// TwinCAT 3 PLC project Simulation_PLC
// ProgramVersion: 3.1.4026.18
// libraries:
//   Tc2_Standard, * (Beckhoff Automation GmbH)
//   Tc2_System, * (Beckhoff Automation GmbH)
//   Tc2_TcpIp, * (Beckhoff Automation GmbH)
//   Tc3_Module, * (Beckhoff Automation GmbH)
// project tree:
//   DUTs/ADS2ROS2/ ST_Pose.TcDUT
//   DUTs/Control/ E_RemoteMode.TcDUT, ST_Control.TcDUT, ST_ControlComau.TcDUT, ST_ControlStewart.TcDUT, ST_ControlWinch.TcDUT
//   DUTs/Feedback/ ST_Feedback.TcDUT, ST_FeedbackComau.TcDUT, ST_FeedbackLeica.TcDUT, ST_FeedbackMru.TcDUT, ST_FeedbackQualisys.TcDUT, ST_FeedbackStewart.TcDUT, ST_FeedbackWinch.TcDUT
//   DUTs/QualisysRT/Components/ ST_3DMarkerPositionNoLabel.TcDUT, ST_3DMarkerPositionNoLabelComponent.TcDUT, ST_RT6D.TcDUT, ST_RT6DComponent.TcDUT, ST_TxHmiQualisys.TcDUT
//   DUTs/QualisysRT/ E_ComponentType.TcDUT, ST_RTComponentData.TcDUT, ST_RTDataQRTPacket.TcDUT
//   DUTs/ ST_RxUdpRemote.TcDUT
//   / PlcTask.TcTTO
//   POUs/ MAIN.TcPOU
//   UDP/ FB_UdpServerRT.TcPOU
// real-time tasks:
//   TASK PlcTask: cycle T#10ms, priority 20, ADS port 350
// I/O:
//   DEVICE Device 1 (EtherCAT), AmsNetId 169.254.119.135.2.1
//     Box 1 (EL6695-0002) [EL6695 EtherCAT Bridge terminal (Secondary)]
//   DEVICE QTM (RT-Ethernet Adapter)
// variable links:
//   Simulation_PLC/Simulation_PLC Instance <-> Device 1 (EtherCAT)/Box 1 (EL6695-0002)
//     PlcTask Inputs/MAIN.nRxCounter <-> IO Inputs/Var 162
//     PlcTask Inputs/MAIN.rxEtherCatBridge <-> IO Inputs/Var 163
//     PlcTask Outputs/MAIN.nTxCounter <-> IO Outputs/Var 164
//     PlcTask Outputs/MAIN.txEtherCatBridge <-> IO Outputs/Var 165

CONFIGURATION Simulation_PLC
    RESOURCE PLC ON TwinCAT3
        TASK PlcTask(INTERVAL := T#10ms, PRIORITY := 20);
        PROGRAM MAIN WITH PlcTask : MAIN;
    END_RESOURCE
END_CONFIGURATION

// ---- DUTs/ADS2ROS2/ST_Pose.TcDUT
TYPE ST_Pose :
STRUCT
	surge : LREAL;
	sway : LREAL;
	heave : LREAL;
	roll : LREAL;
	pitch : LREAL;
	yaw : LREAL;
END_STRUCT
END_TYPE

// ---- DUTs/Control/E_RemoteMode.TcDUT
{attribute 'qualified_only'}
{attribute 'strict'}
{attribute 'to_string'}
TYPE E_RemoteMode :
(
	RemoteUDP,
	RemoteEtherCAT
);
END_TYPE

// ---- DUTs/Control/ST_Control.TcDUT
TYPE ST_Control :
STRUCT
	em8000: ST_ControlStewart;
	em1500: ST_ControlStewart;
	comau: ST_ControlComau;
	winch: ST_ControlWinch;
END_STRUCT
END_TYPE

// ---- DUTs/Control/ST_ControlComau.TcDUT
TYPE ST_ControlComau :
STRUCT
	u : ARRAY[0..5] OF LREAL;

END_STRUCT
END_TYPE

// ---- DUTs/Control/ST_ControlStewart.TcDUT
TYPE ST_ControlStewart :
STRUCT
	// Velocity setpint to stewart
	u : ARRAY[0..5] OF LREAL;
	u_t : ARRAY[0..5] OF LREAL;
	
END_STRUCT
END_TYPE

// ---- DUTs/Control/ST_ControlWinch.TcDUT
TYPE ST_ControlWinch :
STRUCT
	length : LREAL;
	length_t : LREAL;
	length_tt : LREAL;
END_STRUCT
END_TYPE

// ---- DUTs/Feedback/ST_Feedback.TcDUT
TYPE ST_Feedback :
STRUCT
	em8000: ST_FeedbackStewart;
	em1500: ST_FeedbackStewart;
	mru1: ST_FeedbackMru;
	mru2: ST_FeedbackMru;
	comau: ST_FeedbackComau;
	winch: ST_FeedbackWinch;
	qtm: ST_FeedbackQualisys;
	at960: ST_FeedbackLeica;
END_STRUCT
END_TYPE

// ---- DUTs/Feedback/ST_FeedbackComau.TcDUT
TYPE ST_FeedbackComau :
STRUCT
	q: ARRAY[0..5] OF LREAL;
	q_t: ARRAY[0..5] OF LREAL;
END_STRUCT
END_TYPE

// ---- DUTs/Feedback/ST_FeedbackLeica.TcDUT
TYPE ST_FeedbackLeica :
STRUCT
	pos: ARRAY[0..2] OF LREAL;
	R11: LREAL;
	R12: LREAL;
	R13: LREAL;
	R21: LREAL;
	R22: LREAL;
	R23: LREAL;
	R31: LREAL;
	R32: LREAL;
	R33: LREAL;
END_STRUCT
END_TYPE

// ---- DUTs/Feedback/ST_FeedbackMru.TcDUT
TYPE ST_FeedbackMru :
STRUCT
	eta: ARRAY[0..5] OF LREAL;
	v: ARRAY[0..5] OF LREAL;
END_STRUCT
END_TYPE

// ---- DUTs/Feedback/ST_FeedbackQualisys.TcDUT
TYPE ST_FeedbackQualisys :
STRUCT
	dist: LREAL;
	pos: ARRAY[0..2] OF LREAL;
END_STRUCT
END_TYPE

// ---- DUTs/Feedback/ST_FeedbackStewart.TcDUT
TYPE ST_FeedbackStewart :
STRUCT
	eta: ARRAY[0..5] OF LREAL;
	eta_t: ARRAY[0..5] OF LREAL;
	eta_tt: ARRAY[0..5] OF LREAL;
END_STRUCT
END_TYPE

// ---- DUTs/Feedback/ST_FeedbackWinch.TcDUT
TYPE ST_FeedbackWinch :
STRUCT
	length: LREAL;
	length_t: LREAL;
END_STRUCT
END_TYPE

// ---- DUTs/QualisysRT/Components/ST_3DMarkerPositionNoLabel.TcDUT
TYPE ST_3DMarkerPositionNoLabel :
STRUCT
	x : REAL;
	y : REAL;
	z : REAL;
	id : DINT;
END_STRUCT
END_TYPE

// ---- DUTs/QualisysRT/Components/ST_3DMarkerPositionNoLabelComponent.TcDUT
TYPE ST_3DMarkerPositionNoLabelComponent :
STRUCT
	nSize : UDINT;
	nType : UDINT;
	nMarkers : UDINT;
	nDropRate : INT;
	nOutOfSyncRate : INT;
	markers : ARRAY [0..99] OF ST_3DMarkerPositionNoLabel;
END_STRUCT
END_TYPE

// ---- DUTs/QualisysRT/Components/ST_RT6D.TcDUT
TYPE ST_RT6D :
STRUCT
	x : REAL;
	y : REAL;
	z : REAL;
	rotMatrix : ARRAY [0..8] OF REAL;
END_STRUCT
END_TYPE

// ---- DUTs/QualisysRT/Components/ST_RT6DComponent.TcDUT
TYPE ST_RT6DComponent :
STRUCT
	nSize : UDINT;
	nType : UDINT;
	nBodies : UDINT;
	nDropRate : INT;
	nOutOfSyncRate : INT;
	bodies : ARRAY [0..99] OF ST_RT6D;
END_STRUCT
END_TYPE

// ---- DUTs/QualisysRT/Components/ST_TxHmiQualisys.TcDUT
TYPE ST_TxHmiQualisys :
STRUCT
	status : DINT;
	dist : REAL;
	x : REAL;
	y : REAL;
	z : REAL;
	markers : ARRAY [0..9] OF ST_3DMarkerPositionNoLabel;
END_STRUCT
END_TYPE

// ---- DUTs/QualisysRT/E_ComponentType.TcDUT
{attribute 'qualified_only'}
{attribute 'strict'}
TYPE E_ComponentType :
(
	e3D := 1, // 3D marker data
	e3DNoLabel := 2, //Unidentified 3D marker data
	eAnalog := 3, // Analog data from available analog devices
	eForce := 4, // Force data from available force plates.
	e6D := 5, // 6D data - position and rotation matrix
	e6DEuler := 6, // 6D data - position and Euler angles
	e2D := 7, // 2D marker data
	e2DLinearized := 8, // Linearized 2D marker data
	e3DResiduals := 9, // 3D marker data with residuals
 	e3DNoLabelsResiduals := 10, // Unidentified 3D marker data with residuals
	e6DResiduals := 11, // 6D data - position and rotation matrix with residuals
	e6DEulerResiduals := 12, // 6D data - position and Euler angles with residuals
	eAnalogSingle := 13, // Analog data from available analog devices. Only one sample per channel and camera frame. The latest sample is used if more than one sample is available.
	eImage := 14, // Image frame from a specific camera. Image size and format is set with the XML settings, see Image settings.
	eForceSingle := 15 // Force data from available force plates. Only one sample per plate and camera frame. The latest sample is used if more than one sample is available.
);
END_TYPE

// ---- DUTs/QualisysRT/ST_RTComponentData.TcDUT
TYPE ST_RTComponentData :
STRUCT
	nSize : UDINT;
	nType : UDINT;
END_STRUCT
END_TYPE

// ---- DUTs/QualisysRT/ST_RTDataQRTPacket.TcDUT
TYPE ST_RTDataQRTPacket :
STRUCT
	nSize : UDINT;
	nType : UDINT;
	nTimestamp : LINT;
	nFramenumber : UDINT;
	nComponentCount : UDINT;
END_STRUCT
END_TYPE

// ---- DUTs/ST_RxUdpRemote.TcDUT
TYPE ST_RxUdpRemote :
STRUCT
	iUdpKey : UDINT; // Udp Key
	iCounter : UDINT; // Heartbeat counter
	eModeCmd : UDINT; // Operation mode
	em8000_u : ARRAY [0..5] OF REAL; // EM8000 DOF position setpoints
	em8000_u_t : ARRAY [0..5] OF REAL; // EM8000 DOF velocity setpoints
	em1500_u : ARRAY [0..5] OF REAL; // EM1500 DOF position setpoints
	em1500_u_t : ARRAY [0..5] OF REAL; // EM1500 DOF velocity setpoints
	comau_u : ARRAY [0..5] OF REAL; // Joint speed setpoints
	winch_u : REAL; // Winch wire speed setpoint
	
END_STRUCT
END_TYPE

// ---- POUs/MAIN.TcPOU
PROGRAM MAIN
VAR
	// EtherCAT bridge
	rxEtherCatBridge AT %I* : ST_Feedback;
	txEtherCatBridge AT %Q* : ST_Control;
	nRxCounter AT %I* : DINT;
	nTxCounter AT %Q* : DINT;
	nRxCounterOld : DINT;
	
	fTime		: LREAL;
	fDt 		: LREAL := 0.01;
	bEnable		: BOOL := TRUE;
	timer : TON;
	bTimout		 : BOOL;
	
	stEM1500Pose : ST_Pose;
END_VAR

fTime := fTime + fDt;
nTxCounter := nTxCounter + 1;

// ****** Check for timeout ***********
timer.PT := T#500MS;
IF nRxCounter <> nRxCounterOld THEN
    nRxCounterOld := nRxCounter;

    timer(IN := FALSE);
ELSE
    timer(IN := TRUE);
END_IF
bTimout := timer.Q;

stEm1500Pose.surge := rxEtherCatBridge.em1500.eta[0];
stEm1500Pose.sway := rxEtherCatBridge.em1500.eta[1];
stEm1500Pose.heave := rxEtherCatBridge.em1500.eta[2];
stEm1500Pose.roll := rxEtherCatBridge.em1500.eta[3];
stEm1500Pose.pitch := rxEtherCatBridge.em1500.eta[4];
stEm1500Pose.yaw := rxEtherCatBridge.em1500.eta[5];

// --- (optional) legacy sinus test kept for reference ---
// IF bEnable THEN
//     txEtherCatBridge.em1500.u[2] := 0.2*SIN(2.0*3.14*0.1 * fTime);
//     txEtherCatBridge.em8000.u[2] := 0.2*SIN(2.0*3.14*0.1 * fTime);
// ELSE
//     txEtherCatBridge.em1500.u[2] := 0.0;
//     txEtherCatBridge.em8000.u[2] := 0.0;
// END_IF

END_PROGRAM

// ---- UDP/FB_UdpServerRT.TcPOU
{attribute 'c++_compatible'}
FUNCTION_BLOCK FB_UdpServerRT IMPLEMENTS ITcIoUdpProtocolRecv
VAR_INPUT
	
END_VAR
VAR_OUTPUT
	rxBuffer : ARRAY [0..1023] OF BYTE;
END_VAR
VAR
	// ITcIoUdpProtocolRecv related 
	{attribute 'TcInitSymbol'}
	oid : OTCID; 
	ipUdp : ITcIoUdpProtocol;
	
	
	// Initilized variables
	localPort : UINT;
	nRxData : UDINT;
	pRxData : PVOID;
	nTxData : UDINT;
	pTxData : PVOID;
	
	// Remote specification
	remoteIpAddr : UDINT;
	remotePort : UINT;
	
	// Send/Recv counters
	rxCounter : UINT;
	txCounter : UINT;
	
	// Actual rxSize
	rxSize : UDINT;
	
	// Result
	hrInit : HRESULT;
	hrSend : HRESULT;
END_VAR

IF ipUdp <> 0 THEN
	// Check for incoming data
	ipUdp.CheckReceived();
END_IF

{attribute 'conditionalshow'}
METHOD FB_exit : BOOL
VAR_INPUT
	bInCopyCode : BOOL; // if TRUE, the exit method is called for exiting an instance that is copied afterwards (online change).
END_VAR
IF NOT bInCopyCode THEN // no online change
	IF ipUdp <> 0 THEN 
		ipUdp.UnregisterReceiver(localPort); // Shutdown
		FW_SafeRelease(ADR(ipUdp));
		FB_exit := TRUE; 
	END_IF
END_IF
END_METHOD

{attribute 'conditionalshow'}
METHOD FB_init : BOOL
VAR_INPUT
	bInitRetains : BOOL; // if TRUE, the retain variables are initialized (warm start / cold start)
	bInCopyCode : BOOL;  // if TRUE, the instance afterwards gets moved into the copy code (online change)
	
	// Init variables
	_localPort : UINT;
	_nRxData : UDINT;
	_pRxData : PVOID;
	_nTxData : UDINT;
	_pTxData : PVOID;
END_VAR
VAR
    ipSrv : ITComObjectServer;
END_VAR
// Initilize member variables
localPort := _localPort;
nRxData := _nRxData;
pRxData := _pRxData;
nTxData := _nTxData;
pTxData := _pTxData;


IF NOT bInCopyCode THEN // no online change
	IF ipUdp = 0 THEN
	    hrInit := FW_ObjMgr_GetObjectInstance(
			oid:=oid, 
			iid:=TC_GLOBAL_IID_LIST.IID_ITcIoUdpProtocol, 
			pipUnk:=ADR(ipUdp)
		);
		
		IF SUCCEEDED(hrInit) THEN 
			IF  SUCCEEDED(ipUdp.RegisterReceiver(localPort, THIS^)) THEN //open port
				FB_init := TRUE;
			ELSE 
				FW_SafeRelease(ADR(ipUdp));
			END_IF
		END_IF				
	END_IF
END_IF
END_METHOD

{attribute 'conditionalshow'}
METHOD FB_reinit : BOOL
VAR_INPUT
END_VAR
IF (ipUdp <> 0) THEN 
	ipUdp.RegisterReceiver(localPort, THIS^);
	FB_reinit := TRUE; 
END_IF
END_METHOD

{attribute 'object_name' := 'ReceiveData'}
{attribute 'c++_compatible'}
{attribute 'signature_flag' := '33554688'}
{attribute 'pack_mode' := '4'}
{attribute 'show'}
{attribute 'minimal_input_size' := '4'}
METHOD ReceiveData : HRESULT
VAR_INPUT
	ipAddr	: UDINT;
	udpDestPort	: UINT;
	udpSrcPort	: UINT;
	nData	: UDINT;
	pData	: PVOID;
	pVlan	: POINTER TO ETYPE_VLAN_HEADER := 0;
END_VAR
// Read client data
remoteIpAddr := ipAddr;
remotePort := udpSrcPort;

rxCounter := rxCounter + 1;

// Actual size fo data recevied
rxSize := nData;
MEMCPY(ADR(rxBuffer), pData, nData);

IF nData = nRxData THEN
	// Copy recived data
	MEMCPY(pRxData, pData, nRxData);
	
END_IF

IF nTxData > 0 THEN
	// Send data back to client
	hrSend := ipUdp.SendData(ipAddr, udpSrcPort, udpDestPort, nTxData, pTxData, TRUE, 0);
	txCounter := txCounter + 1;
END_IF
END_METHOD

{attribute 'object_name' := 'TcAddRef'}
{attribute 'c++_compatible'}
{attribute 'signature_flag' := '33554688'}
{attribute 'pack_mode' := '4'}
{attribute 'show'}
{attribute 'minimal_input_size' := '4'}
METHOD TcAddRef : UDINT
END_METHOD

{attribute 'object_name' := 'TcQueryInterface'}
{attribute 'c++_compatible'}
{attribute 'signature_flag' := '33554688'}
{attribute 'pack_mode' := '4'}
{attribute 'show'}
{attribute 'minimal_input_size' := '4'}
METHOD TcQueryInterface : HRESULT
VAR_INPUT
	iid	: REFERENCE TO IID;
	pipItf	: POINTER TO PVOID;
END_VAR
VAR
	ipUdpRecv : ITcIoUdpProtocolRecv;
	ipUnknown : ITcUnknown;	
END_VAR
IF GuidsEqual(ADR(iid), ADR(TC_GLOBAL_IID_LIST.IID_ITcIoUdpProtocolRecv)) THEN
	ipUdpRecv := THIS^; // cast to interface pointer
	pipItf^ := ITCUNKNOWN_TO_PVOID(ipUdpRecv);
	TcAddRef();
	TcQueryInterface := S_OK;
ELSIF GuidsEqual(ADR(iid), ADR(TC_GLOBAL_IID_LIST.IID_ITcUnknown)) THEN
	ipUnknown := THIS^; // cast to interface pointer
	pipItf^ := ITCUNKNOWN_TO_PVOID(ipUnknown);
	TcAddRef();
	TcQueryInterface := S_OK;
ELSE
	TcQueryInterface := E_HRESULTAdsErr.NOINTERFACE ; //Call super if this fb extends some other
END_IF
END_METHOD

{attribute 'object_name' := 'TcRelease'}
{attribute 'c++_compatible'}
{attribute 'signature_flag' := '33554688'}
{attribute 'pack_mode' := '4'}
{attribute 'show'}
{attribute 'minimal_input_size' := '4'}
METHOD TcRelease : UDINT
END_METHOD

END_FUNCTION_BLOCK
